// TIA Portal V19 export
TYPE "FCP_STATUS_OUT"
   STRUCT
      FB_Run : Bool := false;
      Reserved_1 : Bool := false;
      Reserved_2 : Bool := false;
      Reserved_3 : Bool := false;
      Mode_24V : Bool := false;
      Sleep_Mode : Bool := false;
      Converter_OK : Bool := false;
      Warning : Bool := false;
      Reserved_8 : Bool := false;
      Reserved_9 : Bool := false;
      Reserved_10 : Bool := false;
      Reserved_11 : Bool := false;
      Slave : Bool := false;
      ParameterGroup1 : Bool := false;
      Vgmin : Bool := false;
      Reserved_15 : Bool := false;
   END_STRUCT;
END_TYPE
